FUNCTION_BLOCK PUBLIC FB_ioSim IMPLEMENTS I_ioInterface
VAR_INPUT
END_VAR
VAR_OUTPUT
END_VAR
VAR
END_VAR

METHOD getOutputs : ST_inputs_analog
getOutputs := P_Simulator.stSimSystemOutputs;
END_METHOD

METHOD setInputs
VAR_INPUT
	stValvePos	: ST_ValvePos;
	eCraneState	: E_CraneStatus;
END_VAR
P_Simulator.stSimInputs := stValvePos;
P_Simulator.eCraneState := eCraneState;
END_METHOD

END_FUNCTION_BLOCK

(* stored: Version 1.1.0.1
   POU FB_ioSim: Id {035cab98-6c47-480f-9cd9-be06721aad9e}, SpecialFunc None
   Method getOutputs: Id {0e518d93-470d-4e93-870a-5c986adabb36}
   Method setInputs: Id {6a353b83-8eef-4c61-9978-024c652f2fc3} *)
